// Mitsubishi GX Works2 project: GX (13)   PLC: FX3G

// global labels: Global1
VAR_GLOBAL
  start_day_switch AT X007 : BOOL;
  indication_light AT X007 : BOOL;
  Y001_coil AT Y001 : BOOL;
  Break_switch AT X002 : BOOL;
  pulse AT X011 : BOOL;
END_VAR
VAR_GLOBAL CONSTANT
  ggggg : REAL := 1000;
END_VAR
VAR_GLOBAL
  bisquit AT D1100 : REAL;
  switch AT X010 : BOOL;
  sen_15 AT X003 : BOOL;
  sen_30 AT X002 : BOOL;
  COIL AT Y004 : BOOL;
  switch1 AT X005 : BOOL;
  help AT M7 : BOOL;
  inventory_pulse AT CS0 : BOOL;
  RE_bisquit AT D1100 : REAL;
  RE_cream AT D1102 : REAL;
  RE_chocolate AT D1104 : REAL;
END_VAR
VAR_GLOBAL CONSTANT
  limit : INT := 6;
  six : INT := 6;
  COnst_6 : REAL := 6;
  COnst_300 : REAL := 300;
END_VAR
VAR_GLOBAL
  helP_2 AT M2 : BOOL;
  switch2 AT X011 : BOOL;
  ziluf_bisquit AT D1110 : REAL;
END_VAR
VAR_GLOBAL CONSTANT
  zillif : INT := 6;
END_VAR
VAR_GLOBAL
  transfer_inv AT X011 : BOOL;
  ziluf_cream AT D1112 : REAL;
END_VAR
VAR_GLOBAL CONSTANT
  zillif6 : REAL := 6;
  zillif300 : REAL := 300;
END_VAR
VAR_GLOBAL
  ziluf_complete AT M3 : BOOL;
  pulse3 AT X007 : BOOL;
  stopper AT TS1 : BOOL;
  timer AT TC1 : BOOL;
END_VAR
VAR_GLOBAL CONSTANT
  TIMER1 : INT := 30;
END_VAR
VAR_GLOBAL
  helP_blink AT M8 : BOOL;
  BLINK_TIMER AT TC4 : BOOL;
END_VAR
VAR_GLOBAL CONSTANT
  TIMER3 : INT := 30;
  TIMER4 : INT := 4;
END_VAR
VAR_GLOBAL
  VALUE_TIMER AT TS4 : BOOL;
  BLINK_COIL AT Y000 : BOOL;
  BLINK_TIMER2 AT TC5 : BOOL;
  VALUE_TIMER5 AT TS5 : BOOL;
  BLINK_COIL2 AT Y001 : BOOL;
  Y007_coil AT Y007 : BOOL;
  B1 AT M12 : BOOL;
END_VAR
VAR_GLOBAL CONSTANT
  TIMER40 : INT := 40;
END_VAR
VAR_GLOBAL
  STOP3 AT TS9 : BOOL;
  pulse12 AT X006 : BOOL;
  analog_input2 AT D8280 : REAL;
  anLOG_INPUT AT D8280 : REAL;
  RE_ANALOG AT D8280 : INT;
  transfer_DATA AT D1120 : INT;
END_VAR
VAR_GLOBAL CONSTANT
  Check : INT := 6;
  CHECK2 : INT := 5;
END_VAR
VAR_GLOBAL
  help14 AT M14 : BOOL;
  reg_cho AT M14 : BOOL;
  DOUBLE_CHO AT M15 : BOOL;
END_VAR
VAR_GLOBAL CONSTANT
  CHOCOLATE : REAL := 120;
END_VAR
VAR_GLOBAL
  TVILA_REGILA : BOOL;
  TVILA AT D1122 : REAL;
END_VAR
VAR_GLOBAL CONSTANT
  aDD23 : REAL := 120;
  aDD2323 : REAL := 240;
END_VAR
VAR_GLOBAL
  COIL123 AT Y003 : BOOL;
  LIGHT AT Y003 : BOOL;
END_VAR
VAR_GLOBAL CONSTANT
  TIMER50 : INT := 50;
END_VAR
VAR_GLOBAL
  switcH0 AT X000 : BOOL;
  firstC AT CC1 : BOOL;
END_VAR
VAR_GLOBAL CONSTANT
  COUNTERK : INT := 5;
END_VAR
VAR_GLOBAL
  OUTC AT CS1 : BOOL;
  COIL_2 AT Y002 : BOOL;
  HELP10 AT M21 : BOOL;
  firstC2 AT CC11 : BOOL;
  firstC23 AT CC11 : BOOL;
END_VAR
VAR_GLOBAL CONSTANT
  COUNTERK6 : INT := 6;
END_VAR
VAR_GLOBAL
  firstC1 AT CC11 : BOOL;
  firstC123 AT CC11 : BOOL;
  TOTAL_CREMBO AT D1124 : INT;
END_VAR
VAR_GLOBAL CONSTANT
  PLUS6 : INT := 6;
  COnst_120 : REAL := 120;
  COnst_240 : REAL := 240;
END_VAR
VAR_GLOBAL
  STOP33 AT TC9 : BOOL;
  STOP_y3 AT TS11 : BOOL;
  STOPY3 AT TC11 : BOOL;
END_VAR
VAR_GLOBAL CONSTANT
  yy : REAL := 6;
  cream300 : REAL := 300;
  bisquit300 : REAL := 6;
  zb6 : REAL := 6;
  zc300 : REAL := 300;
  CHOCOLATE240 : REAL := 240;
END_VAR
VAR_GLOBAL
  COUNTPULSE AT M16 : BOOL;
  Analog AT D8282 : INT;
END_VAR
VAR_GLOBAL CONSTANT
  multiplied : INT := 40;
END_VAR
VAR_GLOBAL
  timer5 AT TS20 : BOOL;
  BLINK_TIMER5 AT TC20 : BOOL;
  Checkkk AT X002 : BOOL;
  helP_30 AT M30 : BOOL;
  z_lamp AT M40 : BOOL;
  z_lamp1 AT M41 : BOOL;
END_VAR
VAR_GLOBAL CONSTANT
  TIMER30 : INT := 30;
END_VAR
VAR_GLOBAL
  STOP30 AT TC21 : BOOL;
  stop_y7 AT TS21 : BOOL;
  helP_blink2 AT M42 : BOOL;
  BLINK_TIMER10 AT TC40 : BOOL;
  VALUE_TIMER2 AT TS40 : BOOL;
  BLINK_TIMER20 AT TC50 : BOOL;
  VALUE_TIMER50 AT TS50 : BOOL;
  touchSensor AT X001 : BOOL;
  touchSensor1 AT X001 : BOOL;
  helP_37 AT M37 : BOOL;
  STOP300 AT TS21 : BOOL;
END_VAR
VAR_GLOBAL CONSTANT
  DIV390 : INT := 390;
END_VAR
VAR_GLOBAL
  help50 AT M50 : BOOL;
END_VAR

// task Task_01 (event TRUE, interval 0, priority 31): POU_01

PROGRAM POU_01
VAR
  B2 : BOOL;
END_VAR
(* structured ladder/FBD written out as ST: instructions are called as NAME(EN, inputs, outputs); _pN, _eN, _tN stand for wires *)
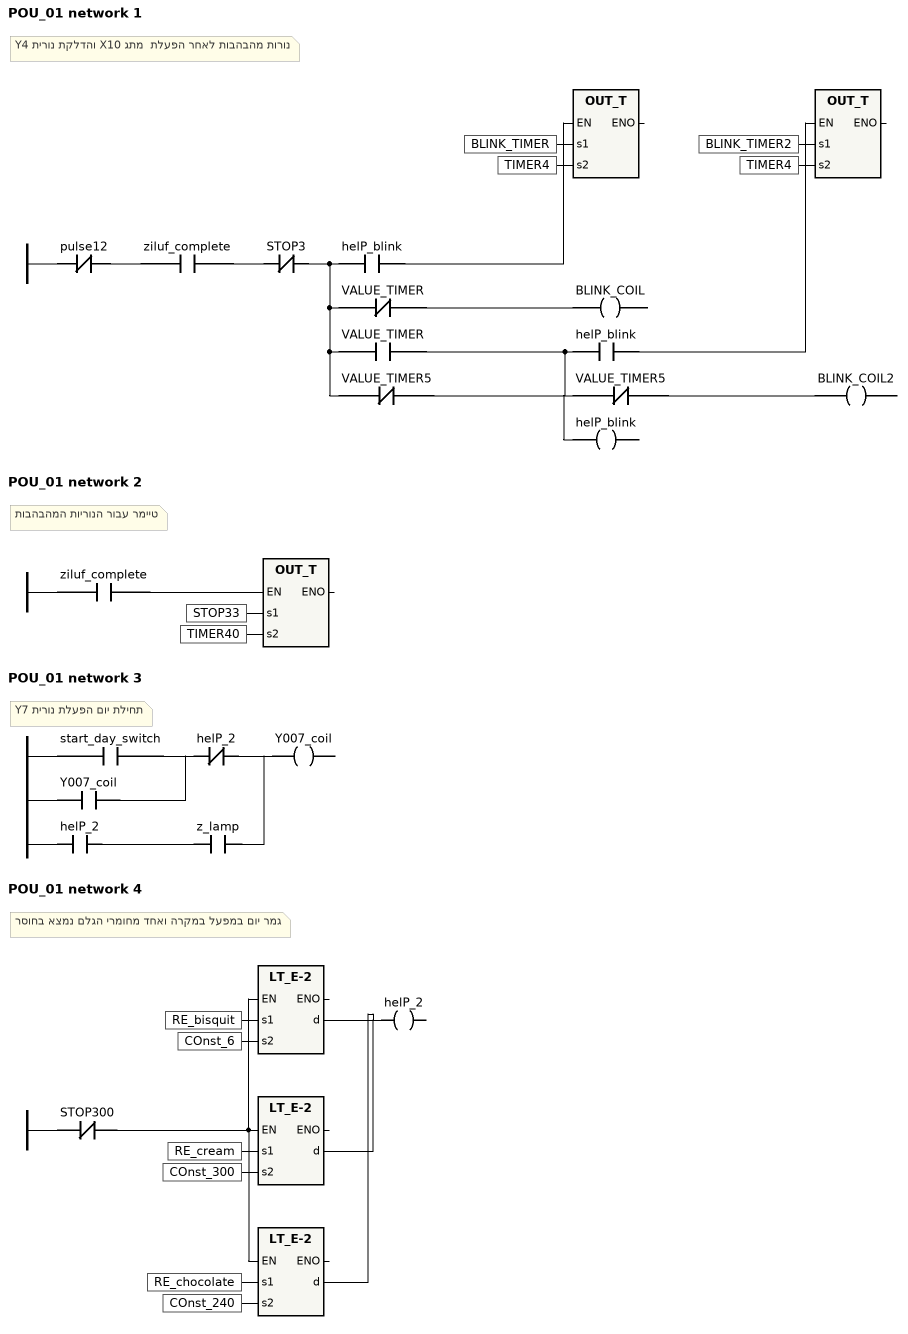
(* network 1 *)
(* נורות מהבהבות לאחר הפעלת  מתג X10 והדלקת נורית Y4 *)
_p1 := NOT pulse12 AND ziluf_complete AND NOT STOP3;
OUT_T(_p1 AND helP_blink, BLINK_TIMER, TIMER4);
BLINK_COIL := _p1 AND NOT VALUE_TIMER;
_p2 := _p1 AND VALUE_TIMER;
OUT_T(_p2 AND helP_blink, BLINK_TIMER2, TIMER4);
BLINK_COIL2 := _p2 AND NOT VALUE_TIMER5;
helP_blink := _p1 AND NOT VALUE_TIMER5;
(* network 2 *)
(* טיימר עבור הנוריות המהבהבות *)
OUT_T(ziluf_complete, STOP33, TIMER40);
(* network 3 *)
(* תחילת יום הפעלת נורית Y7 *)
Y007_coil := ((start_day_switch OR Y007_coil) AND NOT helP_2) OR (helP_2 AND z_lamp);
(* network 4 *)
(* גמר יום במפעל במקרה ואחד מחומרי הגלם נמצא בחוסר *)
_p1 := NOT STOP300;
LT_E(_p1, RE_bisquit, COnst_6, _t2);
LT_E(_p1, RE_cream, COnst_300, _t3);
LT_E(_p1, RE_chocolate, COnst_240, _t4);
helP_2 := _t2 OR _t3 OR _t4;
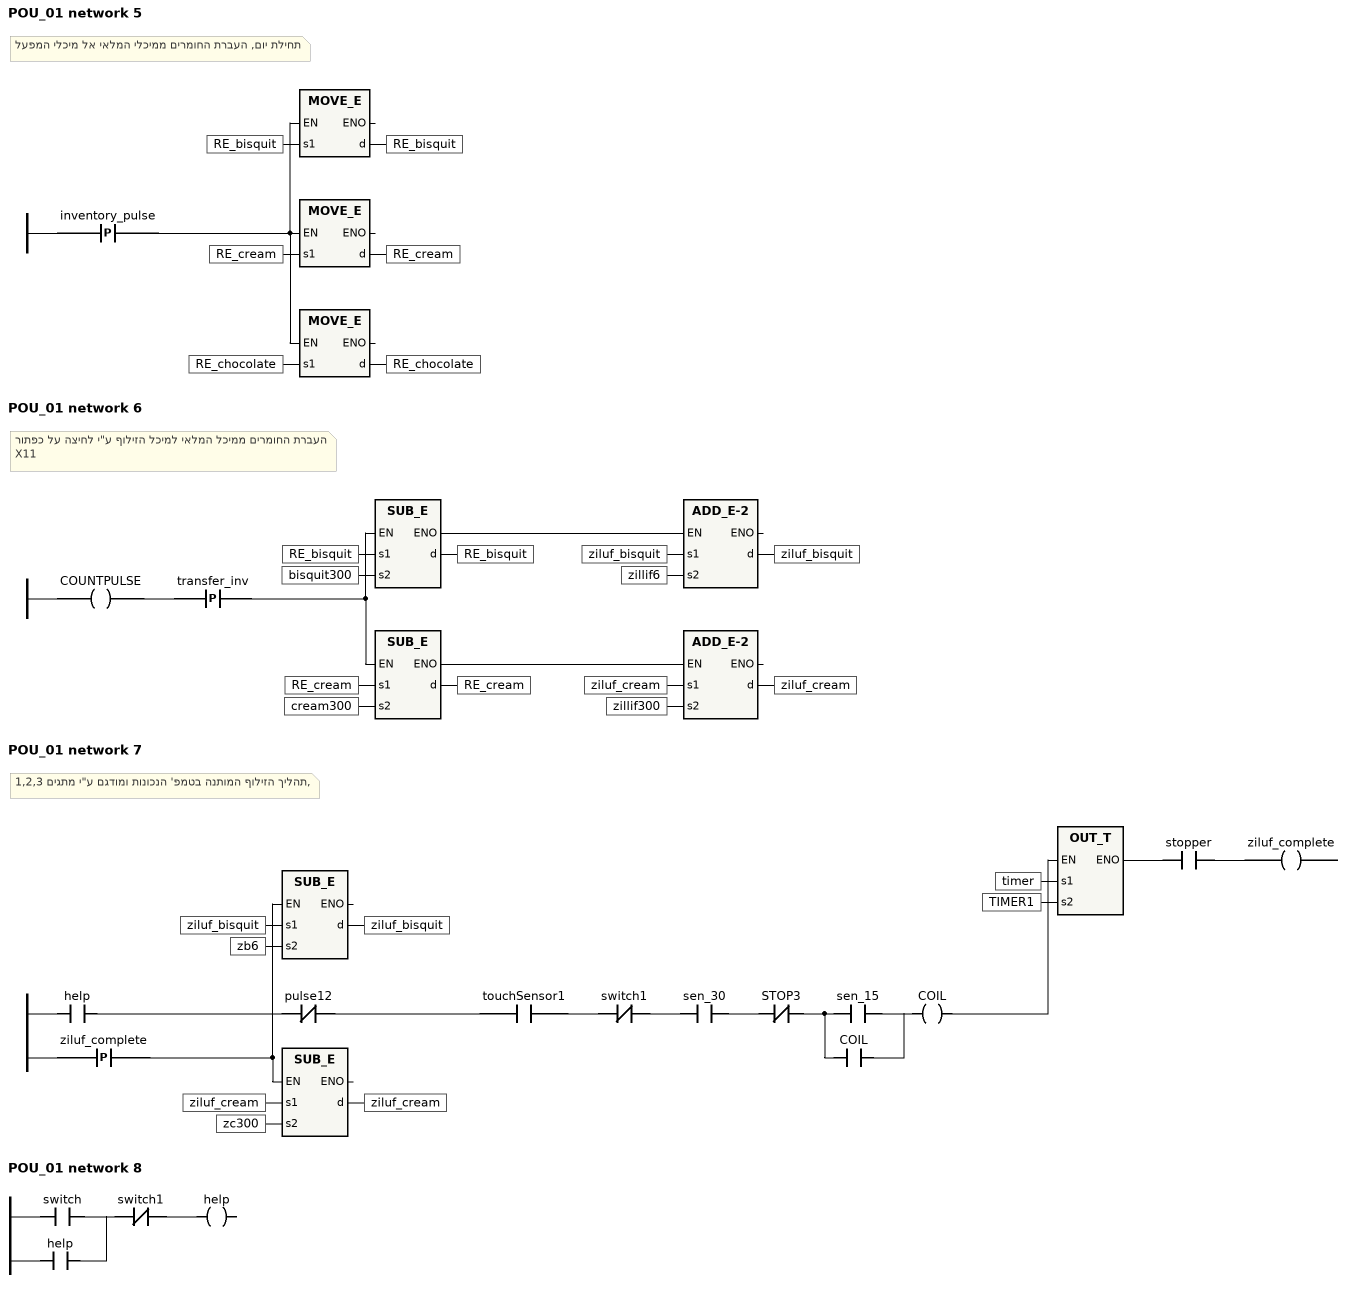
(* network 5 *)
(* תחילת יום, העברת החומרים ממיכלי המלאי אל מיכלי המפעל *)
_p1 := LDP(TRUE, inventory_pulse);
MOVE_E(_p1, RE_bisquit, RE_bisquit);
MOVE_E(_p1, RE_cream, RE_cream);
MOVE_E(_p1, RE_chocolate, RE_chocolate);
(* network 6 *)
(* העברת החומרים ממיכל המלאי למיכל הזילוף ע"י לחיצה על כפתור X11 *)
COUNTPULSE := TRUE;
_p1 := LDP(TRUE, transfer_inv);
_e2 := SUB_E(_p1, RE_bisquit, bisquit300, RE_bisquit);
ADD_E(_e2, ziluf_bisquit, zillif6, ziluf_bisquit);
_e3 := SUB_E(_p1, RE_cream, cream300, RE_cream);
ADD_E(_e3, ziluf_cream, zillif300, ziluf_cream);
(* network 7 *)
(* ,תהליך הזילוף המותנה בטמפ' הנכונות ומודגם ע"י מתגים 1,2,3 *)
_p1 := help AND NOT pulse12 AND touchSensor1 AND NOT switch1 AND sen_30 AND NOT STOP3;
_p2 := (_p1 AND sen_15) OR (_p1 AND COIL);
COIL := _p2;
_e3 := OUT_T(_p2, timer, TIMER1);
ziluf_complete := _e3 AND stopper;
_p4 := LDP(TRUE, ziluf_complete);
SUB_E(_p4, ziluf_bisquit, zb6, ziluf_bisquit);
SUB_E(_p4, ziluf_cream, zc300, ziluf_cream);
(* network 8 *)
help := (switch OR help) AND NOT switch1;
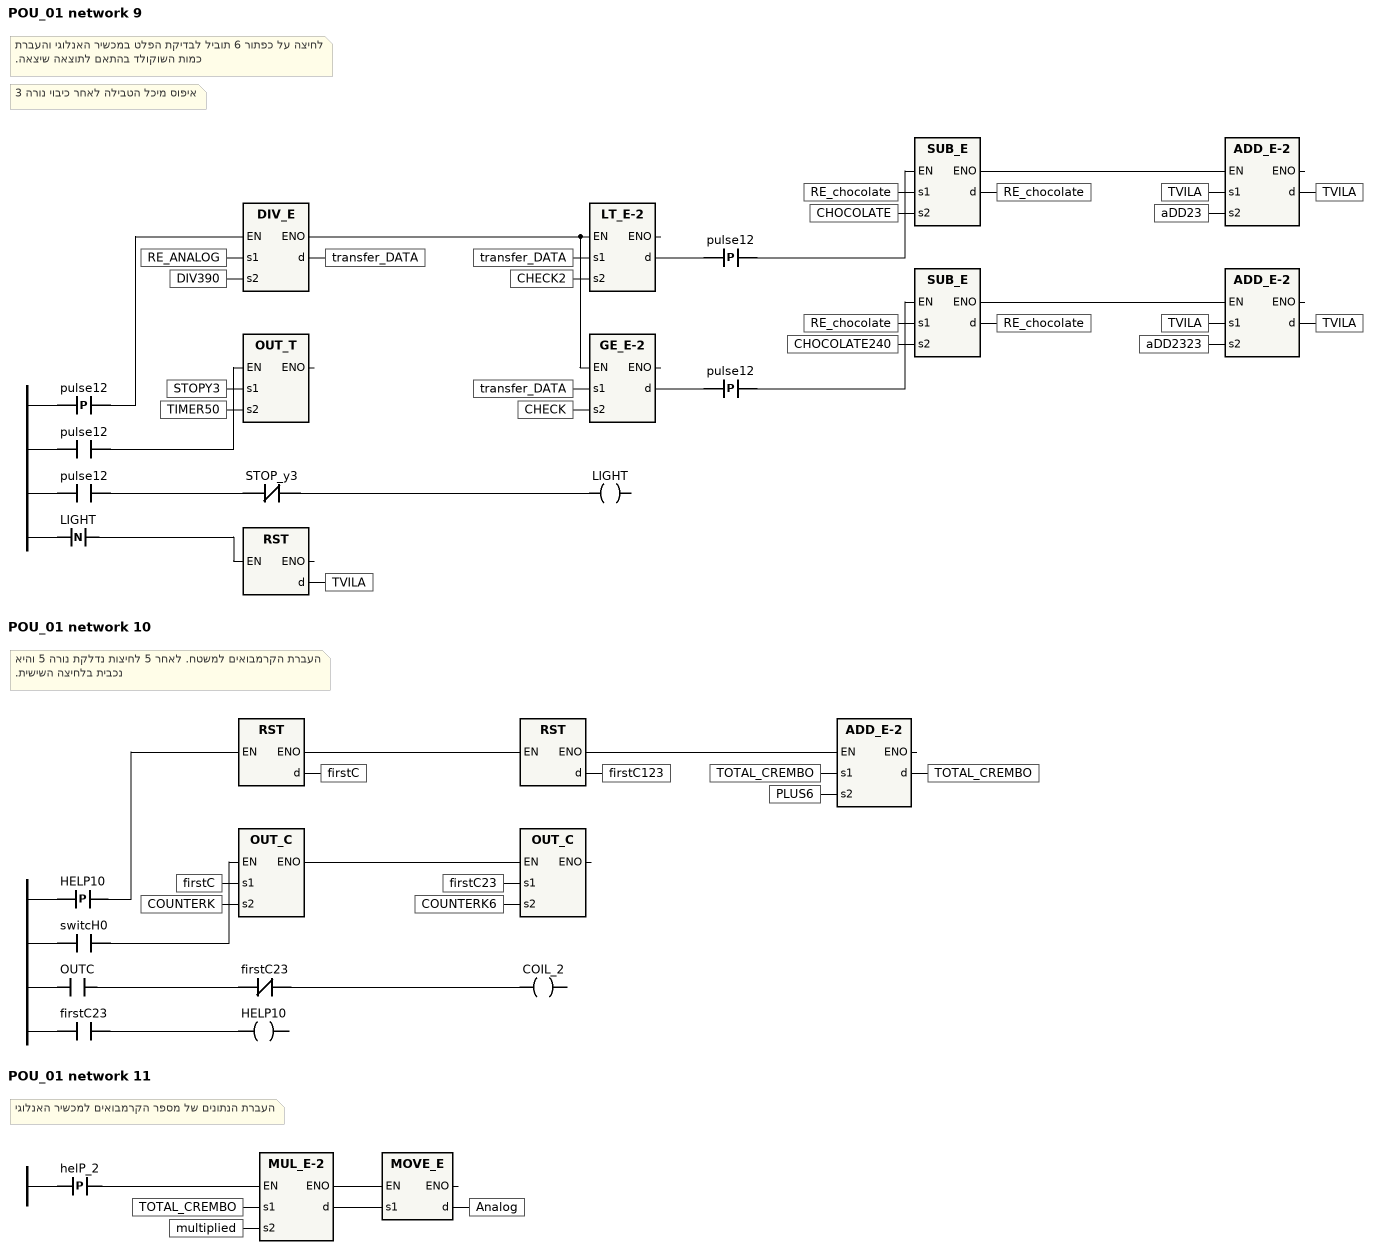
(* network 9 *)
(* לחיצה על כפתור 6 תוביל לבדיקת הפלט במכשיר האנלוגי והעברת כמות השוקולד בהתאם לתוצאה שיצאה. *)
(* איפוס מיכל הטבילה לאחר כיבוי נורה 3 *)
_e1 := DIV_E(LDP(TRUE, pulse12), RE_ANALOG, DIV390, transfer_DATA);
LT_E(_e1, transfer_DATA, CHECK2, _t2);
_e3 := SUB_E(_t2 AND LDP(TRUE, pulse12), RE_chocolate, CHOCOLATE, RE_chocolate);
ADD_E(_e3, TVILA, aDD23, TVILA);
GE_E(_e1, transfer_DATA, CHECK, _t4);
_e5 := SUB_E(_t4 AND LDP(TRUE, pulse12), RE_chocolate, CHOCOLATE240, RE_chocolate);
ADD_E(_e5, TVILA, aDD2323, TVILA);
OUT_T(pulse12, STOPY3, TIMER50);
LIGHT := pulse12 AND NOT STOP_y3;
RST(LDF(TRUE, LIGHT), TVILA);
(* network 10 *)
(* העברת הקרמבואים למשטח. לאחר 5 לחיצות נדלקת נורה 5 והיא נכבית בלחיצה השישית. *)
_e1 := RST(LDP(TRUE, HELP10), firstC);
_e2 := RST(_e1, firstC123);
ADD_E(_e2, TOTAL_CREMBO, PLUS6, TOTAL_CREMBO);
_e3 := OUT_C(switcH0, firstC, COUNTERK);
OUT_C(_e3, firstC23, COUNTERK6);
COIL_2 := OUTC AND NOT firstC23;
HELP10 := firstC23;
(* network 11 *)
(* העברת הנתונים של מספר הקרמבואים למכשיר האנלוגי *)
_e2 := MUL_E(LDP(TRUE, helP_2), TOTAL_CREMBO, multiplied, _t1);
MOVE_E(_e2, _t1, Analog);
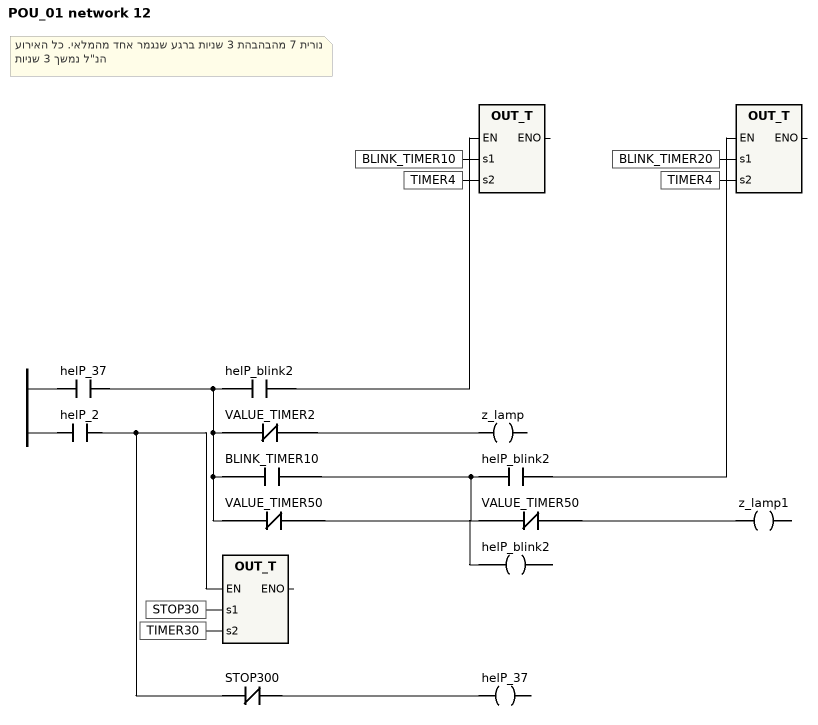
(* network 12 *)
(* נורית 7 מהבהבהת 3 שניות ברגע שנגמר אחד מהמלאי. כל האירוע הנ"ל נמשך 3 שניות *)
OUT_T(helP_37 AND helP_blink2, BLINK_TIMER10, TIMER4);
z_lamp := helP_37 AND NOT VALUE_TIMER2;
_p1 := helP_37 AND BLINK_TIMER10;
OUT_T(_p1 AND helP_blink2, BLINK_TIMER20, TIMER4);
z_lamp1 := _p1 AND NOT VALUE_TIMER50;
helP_blink2 := helP_37 AND NOT VALUE_TIMER50;
OUT_T(helP_2, STOP30, TIMER30);
helP_37 := helP_2 AND NOT STOP300;
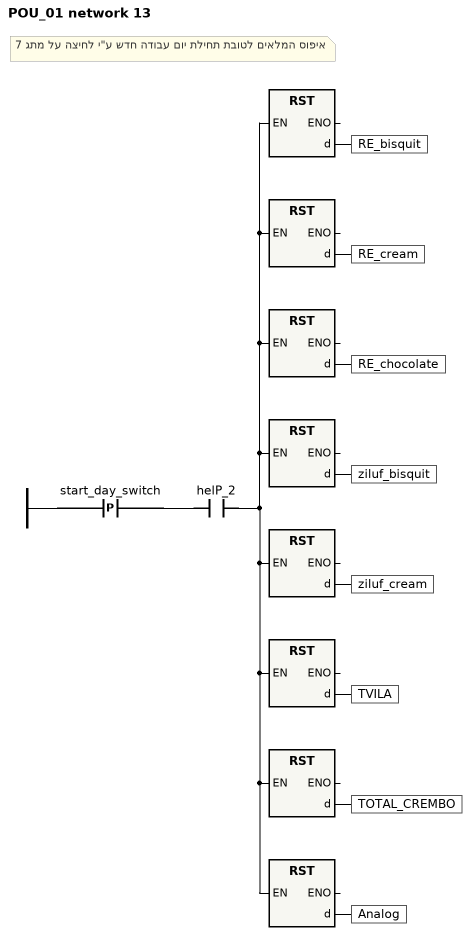
(* network 13 *)
(* איפוס המלאים לטובת תחילת יום עבודה חדש ע"י לחיצה על מתג 7 *)
_p1 := LDP(TRUE, start_day_switch) AND helP_2;
RST(_p1, RE_bisquit);
RST(_p1, RE_cream);
RST(_p1, RE_chocolate);
RST(_p1, ziluf_bisquit);
RST(_p1, ziluf_cream);
RST(_p1, TVILA);
RST(_p1, TOTAL_CREMBO);
RST(_p1, Analog);
END_PROGRAM
